INTERFACE ITF_ObjectExt EXTENDS __System.IQueryInterface

METHOD AddSomeValues : int
VAR_INPUT
	x : INT;
	y : INT;
END_VAR
END_METHOD

END_INTERFACE

(* stored: Version 1.1.0.1, ProductVersion 3.1.4024.11
   Itf ITF_ObjectExt: Id {a93cdcce-2144-4689-9ca6-5b765d666fed}
   Method AddSomeValues: Id {dbf1e4cf-7446-4762-80e1-0768c499d2e9} *)
